ABB RAPID module: RobotTargets.mod

MODULE RobotTargets

    !TEST FOR NOT PULLING FROM RAM

    !CONST robtarget pHeli:=[[-1095.91,2234.75,149.91],[0.00275938,-0.707231,0.706972,-0.00259375],[1,-1,0,0],[0.41674,9E+09,9E+09,9E+09,9E+09,9E+09]];
    CONST robtarget pheli:=[[8943.10,2959.75,271.50],[6.43098E-05,0.707244,-0.706967,-0.00194682],[1,0,0,0],[9020.58,9E+09,9E+09,9E+09,9E+09,9E+09]]; !ax_1 := -230.009
    !Heli pickup
    CONST robtarget pVS:=[[10915.03,2729.72,40.04],[0.00680776,0.00129371,0.999973,0.00247123],[0,-1,0,0],[9402.52,9E+09,9E+09,9E+09,9E+09,9E+09]];
    !VS pickup
    CONST robtarget pPlotter:=[[8711.90,1480.27,-92.24],[7.95004E-05,0.000723003,0.999997,0.00233815],[0,0,0,0],[7000,9E+09,9E+09,9E+09,9E+09,9E+09]];
    !Plotter pickup
    CONST robtarget pHTSHome:=[[-170.79,1515.79,1481.97],[0.00236128,0.676173,-0.736739,0.000524318],[0,0,0,0],[-230.006,9E+09,9E+09,9E+09,9E+09,9E+09]];
    CONST robtarget pVSTSHome:=[[-170.79,1515.79,1481.97],[0.00236128,0.676173,-0.736739,0.000524318],[0,0,0,0],[1200,9E+09,9E+09,9E+09,9E+09,9E+09]];
    CONST robtarget pHeliLid:=[[300,2000,1481.97],[0.00236128,0.676173,-0.736739,0.000524318],[0,0,0,0],[1200,9E+09,9E+09,9E+09,9E+09,9E+09]];
    CONST robtarget pVSLid:=[[-1100,1500,1500],[0.00814298,0.999961,0.000966756,0.00335392],[0,-1,-2,0],[-300,9E+09,9E+09,9E+09,9E+09,9E+09]];

    !CONST robtarget ptHeli:=[[-1090.40,3326.52,-332.42],[0.000292045,-0.707231,0.706978,0.00234295],[1,-1,0,0],[0.419258,9E+09,9E+09,9E+09,9E+09,9E+09]];
    !CONST robtarget ptHeliLid:=[[394.24,3085.52,994.74],[0.00461872,0.67616,-0.736727,-0.00450529],[1,0,0,0],[1200,9E+09,9E+09,9E+09,9E+09,9E+09]];
    CONST robtarget ptHeli:=[[8943.29,2957.80,-354],[6.38917E-05,0.707244,-0.706967,-0.00194727],[1,0,0,0],[9020.58,9E+09,9E+09,9E+09,9E+09,9E+09]];
    CONST robtarget ptHeliLid:=[[394.24,1985.52,994.74],[0.00461872,0.67616,-0.736727,-0.00450529],[1,0,0,0],[1200,9E+09,9E+09,9E+09,9E+09,9E+09]];


    PERS robtarget pTemp;
    VAR robtarget pTemp2;

ENDMODULE
